{attribute 'GeneratedUsingTerminal: EP1809-0042-0019'}
{attribute addProperty BoxType "EP1809-0042-0019"}
{attribute addProperty Description "EP1809-0042 16 Ch. Dig. Input, 3ms, 24 V DC, M12"}
{attribute addProperty Physics "YY"}
{attribute addProperty Id "DI_X01_4AT %I*DI_X_830843C11DI_X01_2AT %I*DI_X_830843C11DI_X02_4AT %I*DI_X_830843C11DI_X02_2AT %I*DI_X_830843C11DI_X03_4AT %I*DI_X_830843C11DI_X03_2AT %I*DI_X_830843C11DI_X04_4AT %I*DI_X_830843C11DI_X04_2AT %I*DI_X_830843C11DI_X05_4AT %I*DI_X_830843C11DI_X05_2AT %I*DI_X_830843C11DI_X06_4AT %I*DI_X_830843C11DI_X06_2AT %I*DI_X_830843C11DI_X07_4AT %I*DI_X_830843C11DI_X07_2AT %I*DI_X_830843C11DI_X08_4AT %I*DI_X_830843C11DI_X08_2AT %I*DI_X_830843C11WcStateAT %I*WcState_9091E0EB2InfoDataAT %I*InfoData_6F19DB2B2"}
{attribute addProperty CRC "2383726614"}
{attribute addProperty Size "20"}
TYPE EP1809_8E14C816 EXTENDS EtcSlaveBoxBase_77A0E4A7 :
STRUCT
	{attribute addProperty Name "DI_X01_4"}
	DI_X01_4 : DI_X_830843C1;
	{attribute addProperty Name "DI_X01_2"}
	DI_X01_2 : DI_X_830843C1;
	{attribute addProperty Name "DI_X02_4"}
	DI_X02_4 : DI_X_830843C1;
	{attribute addProperty Name "DI_X02_2"}
	DI_X02_2 : DI_X_830843C1;
	{attribute addProperty Name "DI_X03_4"}
	DI_X03_4 : DI_X_830843C1;
	{attribute addProperty Name "DI_X03_2"}
	DI_X03_2 : DI_X_830843C1;
	{attribute addProperty Name "DI_X04_4"}
	DI_X04_4 : DI_X_830843C1;
	{attribute addProperty Name "DI_X04_2"}
	DI_X04_2 : DI_X_830843C1;
	{attribute addProperty Name "DI_X05_4"}
	DI_X05_4 : DI_X_830843C1;
	{attribute addProperty Name "DI_X05_2"}
	DI_X05_2 : DI_X_830843C1;
	{attribute addProperty Name "DI_X06_4"}
	DI_X06_4 : DI_X_830843C1;
	{attribute addProperty Name "DI_X06_2"}
	DI_X06_2 : DI_X_830843C1;
	{attribute addProperty Name "DI_X07_4"}
	DI_X07_4 : DI_X_830843C1;
	{attribute addProperty Name "DI_X07_2"}
	DI_X07_2 : DI_X_830843C1;
	{attribute addProperty Name "DI_X08_4"}
	DI_X08_4 : DI_X_830843C1;
	{attribute addProperty Name "DI_X08_2"}
	DI_X08_2 : DI_X_830843C1;
	{attribute addProperty Name "WcState"}
	WcState : WcState_9091E0EB;
	{attribute addProperty Name "InfoData"}
	InfoData : InfoData_6F19DB2B;
END_STRUCT
END_TYPE

(* stored: Version 1.2.0.0, ProductVersion 3.1.4024.11
   DUT EP1809_8E14C816: Id {d92fdaad-7af8-4292-b20b-69f4fc99423a} *)
